(*
	Function block to assign to an ITest interface
*)
{attribute 'NotBlockWritable'}
FUNCTION_BLOCK FB_InterfaceTest IMPLEMENTS ITest
VAR
	(* Last Value *)
	oldValue : BOOL;
END_VAR

(*
	Test method for the ITest interface
*)
METHOD TestMethod : BOOL	(* Inverted value since last call *)
(* Return the inverted old value and save the inverted value as the new old value *)
TestMethod := NOT oldValue;
oldValue := TestMethod;
END_METHOD

END_FUNCTION_BLOCK

(* stored: Version 1.1.0.1
   POU FB_InterfaceTest: Id {28fe76e9-abf0-41b4-92c9-4dc26c68cb8e}, SpecialFunc None
   Method TestMethod: Id {1f73adbc-99da-4c1f-a591-4c55a32e74c2} *)
